SUBAPPLICATION AR_R_MUL (* Multipliziert einen AR-Wert mit einem festen REAL-Faktor (kein zweiter AR-Socket noetig - der Faktor wird per Parameter bei der Instanziierung eingebacken) *)
  (* Standard: 61499-2 *)
  (* Version 1.0, 2026-09-08, Franz Höpfinger, Meisterschulen am Ostbahnhof *)
  PACKAGE MyLib::sys;
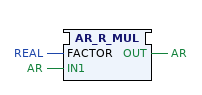
  VAR_INPUT
    FACTOR : REAL := REAL#1.0; (* Fester Multiplikator, ueber Parameter bei der Instanziierung gesetzt *)
  END_VAR
  SOCKETS
    IN1 : adapter::types::unidirectional::AR; (* Zu skalierender Wert *)
  END_SOCKETS
  PLUGS
    OUT : adapter::types::unidirectional::AR; (* IN1 x FACTOR *)
  END_PLUGS
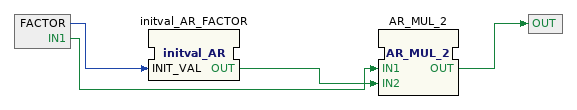
  FBS
    initval_AR_FACTOR : adapter::types::unidirectional::AR::initval::initval_AR;
    AR_MUL_2 : adapter::iec61131::arithmetic::AR_MUL_2;
  END_FBS
  DATA_CONNECTIONS
    FACTOR TO initval_AR_FACTOR.INIT_VAL;
  END_CONNECTIONS
  ADAPTER_CONNECTIONS
    IN1 TO AR_MUL_2.IN1;
    initval_AR_FACTOR.OUT TO AR_MUL_2.IN2;
    AR_MUL_2.OUT TO OUT;
  END_CONNECTIONS
END_SUBAPPLICATION
